(* PLC project Unnamed, Unknown Unnamed 1 *)
(* stored: creationDateTime 2026-04-16T13:53:00, modificationDateTime 2026-04-16T13:53:00 *)

PROGRAM main
  VAR
    sensor_temp AT %MW0 : INT;
    fan_speed AT %QW0 : INT;
    sensor_power AT %MW1 : INT;
    overheat_alarm AT %QX0.0 : BOOL;
  END_VAR
  VAR
    CRAC_Fan_Status : BOOL;
    Temp_High_Alarm : BOOL;
  END_VAR

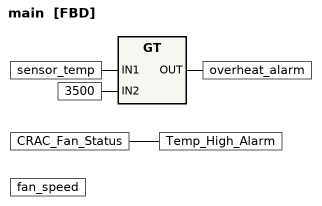
(* FBD diagram, written out as Structured Text *)
Temp_High_Alarm := CRAC_Fan_Status;
overheat_alarm := sensor_temp > 3500;
END_PROGRAM

CONFIGURATION Config0
  RESOURCE Res0 ON PLC
    TASK task0(INTERVAL := T#20ms, PRIORITY := 1);
    PROGRAM instance0 WITH task0 : main;
  END_RESOURCE
END_CONFIGURATION
